INTERFACE I_PathAStarNode EXTENDS I_CH_Object

{attribute 'monitoring':='call'}
PROPERTY PathLength : LREAL
GET
END_GET
END_PROPERTY

{attribute 'monitoring':='call'}
PROPERTY RouteUsedToNode : REFERENCE TO FB_CH_List
GET
END_GET
END_PROPERTY

{attribute 'monitoring':='call'}
PROPERTY Station : I_XP_Station
GET
END_GET
SET
END_SET
END_PROPERTY

END_INTERFACE

(* stored: Version 1.1.0.1, ProductVersion 3.1.4024.12
   Itf I_PathAStarNode: Id {be03b726-bf5e-4aa4-8cbd-e6818b63cc5e}
   Property PathLength: Id {a1e7f472-e25c-4988-874a-405294be83bf}
   Get Get: Id {402d665a-0db6-41d8-9d96-effb115101f5}
   Property RouteUsedToNode: Id {cf4d0ab7-cd67-48fa-9114-196361431315}
   Get Get: Id {a132d470-0dc2-4e7d-90e1-0fc70318764b}
   Property Station: Id {40b98fe3-6617-45bb-859c-69640d2a05e6}
   Get Get: Id {8f793438-1b54-4ae9-a9ba-6b113472ffc5}
   Set Set: Id {fae487dc-535b-45a1-a0f9-4ba413d05a38} *)
